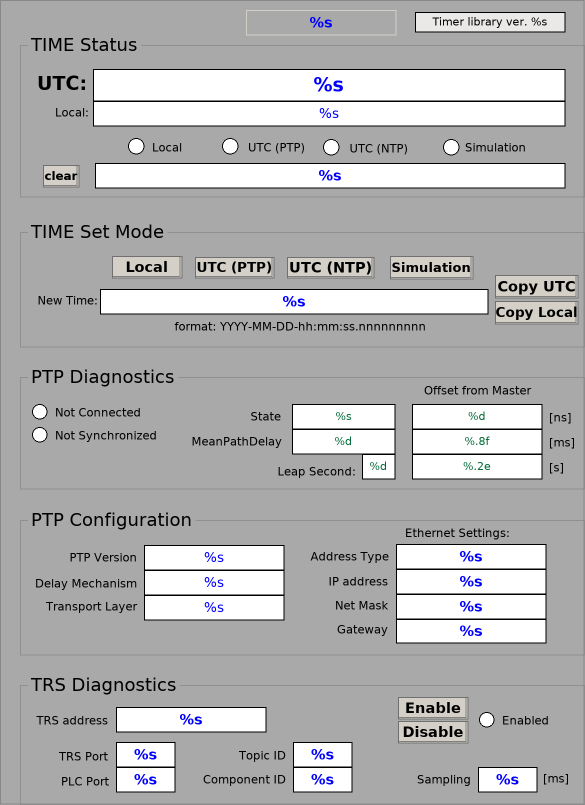
VISUALIZATION GUI_TEMPLATE_TIME  // 585x805
VAR_INPUT
	m_DeviceName : STRING;
END_VAR
VAR_IN_OUT
	m_Instance : FB_TIME;
END_VAR
    GroupBox (20,369 565x120), "PTP Diagnostics"
        Label (391,10 133x23), "Offset from Master"
        Rectangle (272,35 103x25), "%s", text variable: m_Instance.stat.el6688.diagnostics.ptp_state
        Label (222,35 42x25), "State"
        Label (229,90 110x25), "Leap Second:"
        Rectangle (342,85 33x25), "%d", text variable: m_Instance.stat.el6688.diagnostics.leap_second
        Rectangle (392,35 130x25), "%d", text variable: m_Instance.stat.el6688.diagnostics.offset_from_master
        Label (526,35 31x27), "[ns]"
        Rectangle (392,85 130x25), "%.2e", text variable: m_Instance.stat.el6688.diagnostics.offset_from_master_sec
        Label (526,60 31x27), "[ms]"
        Label (526,85 20x27), "[s]"
        Rectangle (392,60 130x25), "%.8f", text variable: m_Instance.stat.el6688.diagnostics.offset_from_master_msec
        Ellipse (12,35 15x15), tooltip "WHITE=Connected RED=Not Connected", colour toggle: (m_Instance.stat.signal.status) = E_TIME_SIGNAL_STATUS.NOT_CONNECTED
        Ellipse (12,58 15x15), tooltip "WHITE=Synchronized RED=Not Synchronized", colour toggle: (m_Instance.stat.signal.qos) = E_TIME_SIGNAL_QOS.NOT_SYNCHRONIZED
        Label (32,31 97x25), "Not Connected"
        Label (32,54 106x25), "Not Synchronized"
        Label (166,60 99x25), "MeanPathDelay"
    GroupBox (20,37 565x160), "TIME Status"
        Label (23,61 49x29), "Local:"
        Label (113,98 52x25), "Local"
        Rectangle (73,64 472x25), "%s", text variable: m_Instance.stat.sDcTime
        Rectangle (73,32 472x32), "%s", text variable: m_Instance.stat.sUtcTime
        Rectangle (75,126 470x25), "%s", tooltip "Error Message", text variable: m_Instance.stat.sErrorMsg
        Ellipse (108,101 16x16), tooltip "Active time: Local", colour toggle: (m_Instance.stat.mode) = E_TIME_MODE.LOCAL
        Ellipse (202,101 16x16), tooltip "Active time: UTC", colour toggle: (m_Instance.stat.mode = E_TIME_MODE.UTC_PTP)
        Ellipse (423,102 16x16), tooltip "Active time: Simulated", colour toggle: (m_Instance.stat.mode) = E_TIME_MODE.SIMULATION
        Label (430,98 79x25), "Simulation"
        Label (217,98 71x25), "UTC (PTP)"
        Label (321,99 70x25), "UTC (NTP)"
        Ellipse (303,102 16x16), tooltip "Active time: UTC", colour toggle: (m_Instance.stat.mode = E_TIME_MODE.UTC_NTP)
        Button (23,128 36x22), "clear", tooltip "Use local time"
            OnMouseClick: execute { m_Instance.stat.sErrorMsg := ''; }
    GroupBox (20,512 565x143), "PTP Configuration"
        Label (281,80 90x27), "Net Mask"
        Rectangle (376,57 150x25), "%s", text variable: m_Instance.stat.el6688.config.ethernet_settings.ip_address
        Rectangle (376,82 150x25), "%s", text variable: m_Instance.stat.el6688.config.ethernet_settings.subnet_mask
        Label (34,32 86x27), "PTP Version"
        Label (281,105 90x25), "Gateway"
        Rectangle (124,33 140x25), "%s", text variable: m_Instance.stat.el6688.config.ptp_version
        Label (352,7 141x28), "Ethernet Settings:"
        Rectangle (376,107 150x24), "%s", text variable: m_Instance.stat.el6688.config.ethernet_settings.gateway
        Label (7,58 113x27), "Delay Mechanism"
        Rectangle (124,58 140x25), "%s", text variable: m_Instance.stat.el6688.config.delay_mechanism
        Label (10,81 110x27), "Transport Layer"
        Rectangle (376,32 150x25), "%s", text variable: m_Instance.stat.el6688.config.ethernet_settings.address_type
        Rectangle (124,83 140x25), "%s", text variable: m_Instance.stat.el6688.config.transport_layer
        Label (282,30 90x29), "Address Type"
        Label (281,55 90x29), "IP address"
    Label (9,68 81x31), "UTC:"
    Rectangle (246,10 150x25), "%s", text variable: m_DeviceName
    Rectangle (415,12 150x20), "Timer library ver. %s", text variable: m_Instance.stat.sLibVersion
    GroupBox (20,224 565x123), "TIME Set Mode"
        Button (92,32 70x22), "Local", tooltip "Use local time"
            OnMouseClick: execute { m_Instance.cfg.nMode := E_TIME_MODE.LOCAL; }
        Button (175,33 79x21), "UTC (PTP)", tooltip "Use UTC time (source PTP)"
            OnMouseClick: execute { m_Instance.cfg.nMode := E_TIME_MODE.UTC_PTP; }
        Rectangle (80,65 388x25), "%s", tooltip "Time used for Simulation. Press "Copy UTC" or "Copy Local" button to get the time in correct format and then modify it for your needs.", text variable: m_Instance.cfg.sUserTime
            OnMouseDown: write the text variable via Default
        Button (370,32 83x23), "Simulation", tooltip "Use simulated time given under "New Time". NOTE: "New Time" is taken only if the time string has been modified since the last press of the button."
            OnMouseClick: execute { m_Instance.cfg.nMode := E_TIME_MODE.SIMULATION; }
        Label (8,64 73x25), "New Time:"
        Label (139,90 270x25), "format: YYYY-MM-DD-hh:mm:ss.nnnnnnnnn"
        Button (475,51 83x23), "Copy UTC", tooltip "Copy current UTC time to "New Time""
            OnMouseClick: execute { m_Instance.cfg.sUserTime := m_Instance.stat.sUtcTime; }
        Button (267,33 87x21), "UTC (NTP)", tooltip "Use UTC time ((source NTP)"
            OnMouseClick: execute { m_Instance.cfg.nMode := E_TIME_MODE.UTC_NTP; }
    GroupBox (20,677 565x128), "TRS Diagnostics"
        Rectangle (96,65 59x25), "%s", text variable: m_Instance.cfg.diag_report.destination_port
            OnMouseDown: write the text variable via Edit
        Button (378,20 70x22), "Enable", tooltip "Enable Diagnostics"
            OnMouseClick: execute { m_Instance.cfg.diag_report.enabled := TRUE; }
        Button (378,44 70x22), "Disable", tooltip "Disable Diagnostics"
            OnMouseClick: execute { m_Instance.cfg.diag_report.enabled := FALSE; }
        Rectangle (96,90 59x25), "%s", text variable: m_Instance.cfg.diag_report.source_port
            OnMouseDown: write the text variable via Edit
        Label (7,29 84x29), "TRS address"
        Label (479,29 61x29), "Enabled"
        Label (32,65 59x29), "TRS Port"
        Label (23,90 69x29), "PLC Port"
        Label (387,88 67x29), "Sampling"
        Label (521,88 31x27), "[ms]"
        Rectangle (458,90 59x25), "%s", text variable: m_Instance.cfg.diag_report.sampling
            OnMouseDown: write the text variable via Edit
        Ellipse (459,35 15x15), tooltip "WHITE - Disabled GREEN - Enabled", colour toggle: m_Instance.stat.diag_report.enabled
        Rectangle (96,30 150x25), "%s", text variable: m_Instance.cfg.diag_report.address
            OnMouseDown: write the text variable via Edit
        Rectangle (273,65 59x25), "%s", text variable: m_Instance.cfg.diag_report.topic_id
            OnMouseDown: write the text variable via Edit
        Label (210,64 59x29), "Topic ID"
        Label (182,88 87x29), "Component ID"
        Rectangle (273,90 59x25), "%s", text variable: m_Instance.cfg.diag_report.compontent_id
            OnMouseDown: write the text variable via Edit
    Button (495,301 83x23), "Copy Local", tooltip "Copy current Local time to "New Time""
        OnMouseClick: execute { m_Instance.cfg.sUserTime := m_Instance.stat.sDcTime; }
    Rectangle (292,429 103x25), "%d", text variable: m_Instance.stat.el6688.diagnostics.mean_path_delay
END_VISUALIZATION

(* stored: Version 1.1.0.1, ProductVersion 3.1.4024.11
   Visu GUI_TEMPLATE_TIME: Id {9265c798-38b0-452a-bfbb-7e96b4d7ae66} *)
